% RSLogix 500 project Complex Boiler System.RSS, saved by version 8.30.00.16 %
PROJECT "UNTITLED"    % processor: Bul.1763 MicroLogix 1100 Series B %

PROGRAM FILES
  LAD 2 "MAIN"  10 rungs
  LAD 3 "DIGI IN"  11 rungs  % Digital Input Ladder Logic %
  LAD 4 "DIGI OUT"  4 rungs  % Digital Output Ladder Logic %
  LAD 5 "ANALOG IN"  5 rungs  % Analog Inout Ladder Logic %
  LAD 6 "ANALOG OUT"  2 rungs  % Analog Output Ladder Logic %
  LAD 7 "CONTROLS"  15 rungs
  LAD 8 "ALARMS"  28 rungs
  LAD 9 "DISPLAY"  2 rungs

DATA FILES
  O0 OUTPUT  9 elements
  I1 INPUT  16 elements
  S2 STATUS  66 elements
  B3 BINARY  5 elements
  T4 TIMER  13 elements
  C5 COUNTER  1 elements
  R6 CONTROL  1 elements
  N7 INTEGER  9 elements
  F8 FLOAT  1 elements
  PD9   1 elements

LADDER 2 "MAIN"
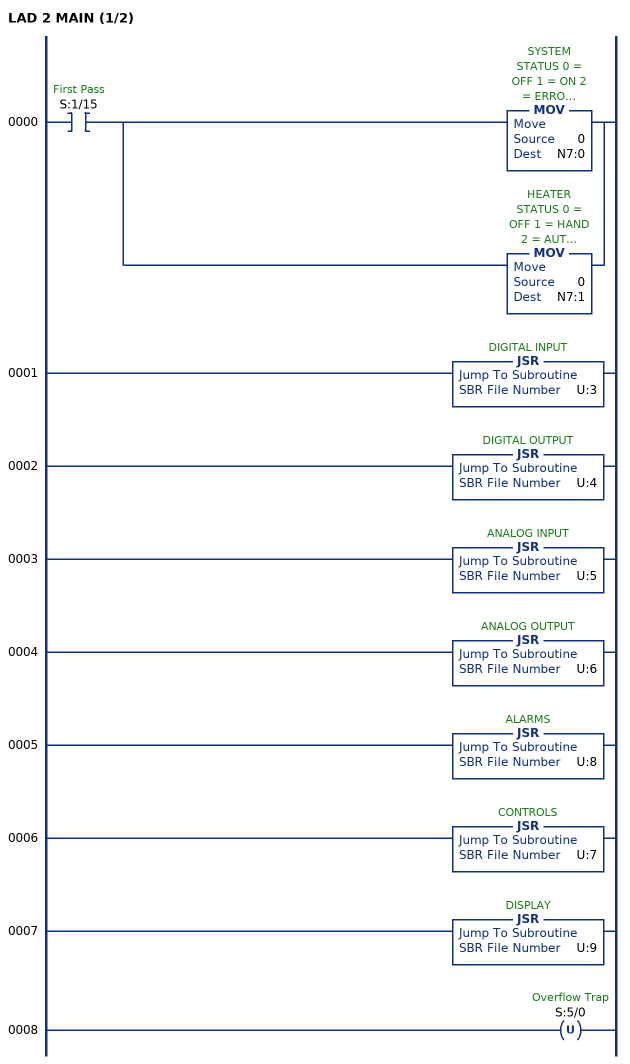
% Rung: 0 %
SOR XIC S:1/15 BST MOV 0 N7:0 NXB MOV 0 N7:1 BND EOR
%   S:1/15  "First Pass" %
%   N7:0  SYSTEM_STATUS  "SYSTEM STATUS 0 = OFF 1 = ON 2 = ERROR" %
%   N7:1  HEATER_STATUS  "HEATER STATUS 0 = OFF 1 = HAND 2 = AUTO" %
% Rung: 1 %
SOR JSR U:3 EOR
%   U:3  "DIGITAL INPUT" %
% Rung: 2 %
SOR JSR U:4 EOR
%   U:4  "DIGITAL OUTPUT" %
% Rung: 3 %
SOR JSR U:5 EOR
%   U:5  "ANALOG INPUT" %
% Rung: 4 %
SOR JSR U:6 EOR
%   U:6  "ANALOG OUTPUT" %
% Rung: 5 %
SOR JSR U:8 EOR
%   U:8  "ALARMS" %
% Rung: 6 %
SOR JSR U:7 EOR
%   U:7  "CONTROLS" %
% Rung: 7 %
SOR JSR U:9 EOR
%   U:9  "DISPLAY" %
% Rung: 8 %
SOR OTU S:5/0 EOR
%   S:5/0  "Overflow Trap" %

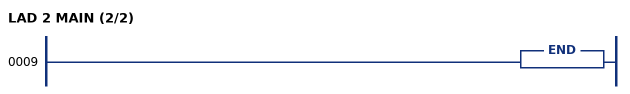
% Rung: 9 %
SOR END EOR

LADDER 3 "DIGI IN"    % Digital Input Ladder Logic %
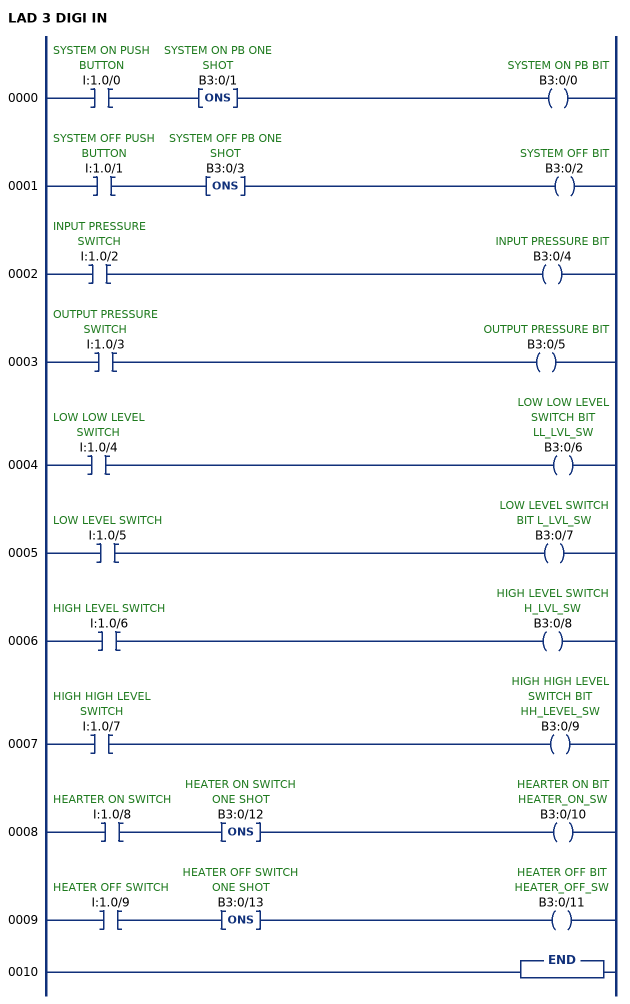
% Rung: 0 %
SOR XIC I:1.0/0 ONS B3:0/1 OTE B3:0/0 EOR
%   I:1.0/0  "SYSTEM ON PUSH BUTTON" %
%   B3:0/1  "SYSTEM ON PB ONE SHOT" %
%   B3:0/0  "SYSTEM ON PB BIT" %
% Rung: 1 %
SOR XIC I:1.0/1 ONS B3:0/3 OTE B3:0/2 EOR
%   I:1.0/1  "SYSTEM OFF PUSH BUTTON" %
%   B3:0/3  "SYSTEM OFF PB ONE SHOT" %
%   B3:0/2  "SYSTEM OFF BIT" %
% Rung: 2 %
SOR XIC I:1.0/2 OTE B3:0/4 EOR
%   I:1.0/2  "INPUT PRESSURE SWITCH" %
%   B3:0/4  "INPUT PRESSURE BIT" %
% Rung: 3 %
SOR XIC I:1.0/3 OTE B3:0/5 EOR
%   I:1.0/3  "OUTPUT PRESSURE SWITCH" %
%   B3:0/5  "OUTPUT PRESSURE BIT" %
% Rung: 4 %
SOR XIC I:1.0/4 OTE B3:0/6 EOR
%   I:1.0/4  "LOW LOW LEVEL SWITCH" %
%   B3:0/6  LL_LVL_SW  "LOW LOW LEVEL SWITCH BIT" %
% Rung: 5 %
SOR XIC I:1.0/5 OTE B3:0/7 EOR
%   I:1.0/5  "LOW LEVEL SWITCH" %
%   B3:0/7  L_LVL_SW  "LOW LEVEL SWITCH BIT" %
% Rung: 6 %
SOR XIC I:1.0/6 OTE B3:0/8 EOR
%   I:1.0/6  "HIGH LEVEL SWITCH" %
%   B3:0/8  H_LVL_SW  "HIGH LEVEL SWITCH" %
% Rung: 7 %
SOR XIC I:1.0/7 OTE B3:0/9 EOR
%   I:1.0/7  "HIGH HIGH LEVEL SWITCH" %
%   B3:0/9  HH_LEVEL_SW  "HIGH HIGH LEVEL SWITCH BIT" %
% Rung: 8 %
SOR XIC I:1.0/8 ONS B3:0/12 OTE B3:0/10 EOR
%   I:1.0/8  "HEARTER ON SWITCH" %
%   B3:0/12  "HEATER ON SWITCH ONE SHOT" %
%   B3:0/10  HEATER_ON_SW  "HEARTER ON BIT" %
% Rung: 9 %
SOR XIC I:1.0/9 ONS B3:0/13 OTE B3:0/11 EOR
%   I:1.0/9  "HEATER OFF SWITCH" %
%   B3:0/13  "HEATER OFF SWITCH ONE SHOT" %
%   B3:0/11  HEATER_OFF_SW  "HEATER OFF BIT" %
% Rung: 10 %
SOR END EOR

LADDER 4 "DIGI OUT"    % Digital Output Ladder Logic %
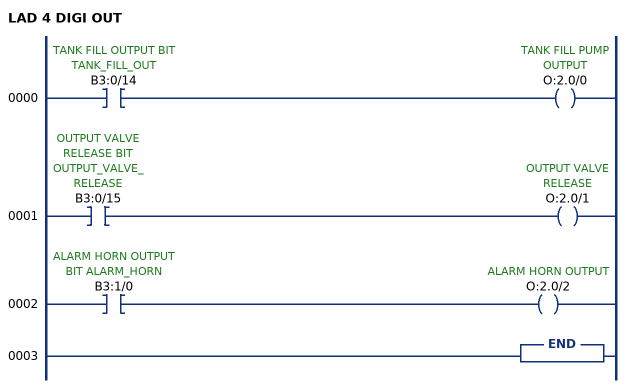
% Rung: 0 %
SOR XIC B3:0/14 OTE O:2.0/0 EOR
%   B3:0/14  TANK_FILL_OUT  "TANK FILL OUTPUT BIT" %
%   O:2.0/0  "TANK FILL PUMP OUTPUT" %
% Rung: 1 %
SOR XIC B3:0/15 OTE O:2.0/1 EOR
%   B3:0/15  OUTPUT_VALVE_RELEASE  "OUTPUT VALVE RELEASE BIT" %
%   O:2.0/1  "OUTPUT VALVE RELEASE" %
% Rung: 2 %
SOR XIC B3:1/0 OTE O:2.0/2 EOR
%   B3:1/0  ALARM_HORN  "ALARM HORN OUTPUT BIT" %
%   O:2.0/2  "ALARM HORN OUTPUT" %
% Rung: 3 %
SOR END EOR

LADDER 5 "ANALOG IN"    % Analog Inout Ladder Logic %
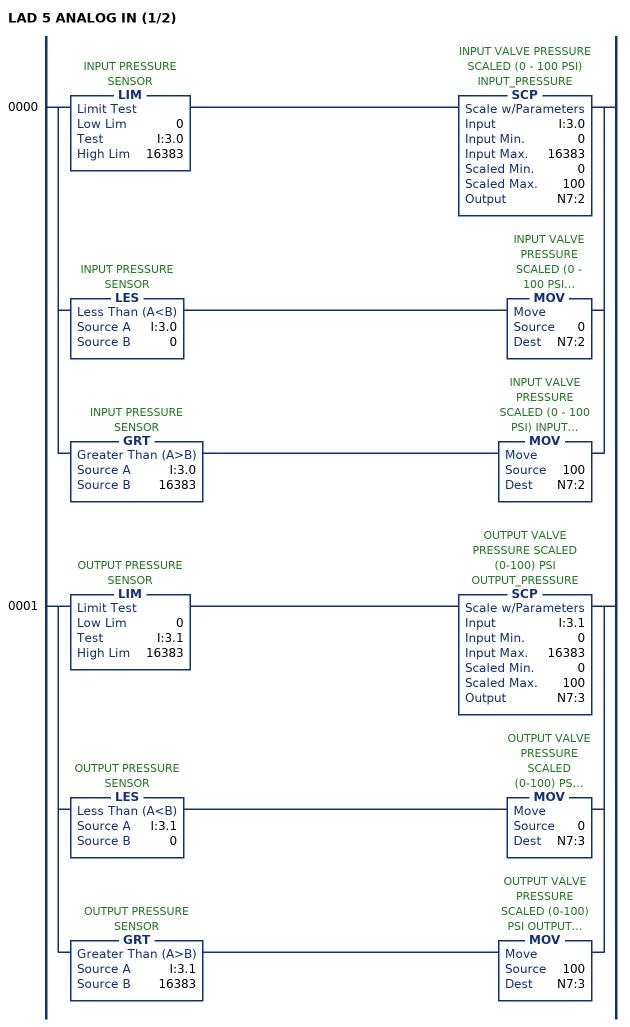
% Rung: 0 %
SOR BST LIM 0 I:3.0 16383 SCP I:3.0 0 16383 0 100 N7:2 NXB LES I:3.0 0 MOV 0 N7:2 NXB GRT I:3.0 16383 MOV 100 N7:2 BND EOR
%   I:3.0  "INPUT PRESSURE SENSOR" %
%   N7:2  INPUT_PRESSURE  "INPUT VALVE PRESSURE SCALED (0 - 100 PSI)" %
% Rung: 1 %
SOR BST LIM 0 I:3.1 16383 SCP I:3.1 0 16383 0 100 N7:3 NXB LES I:3.1 0 MOV 0 N7:3 NXB GRT I:3.1 16383 MOV 100 N7:3 BND EOR
%   I:3.1  "OUTPUT PRESSURE SENSOR" %
%   N7:3  OUTPUT_PRESSURE  "OUTPUT VALVE PRESSURE SCALED (0-100) PSI" %

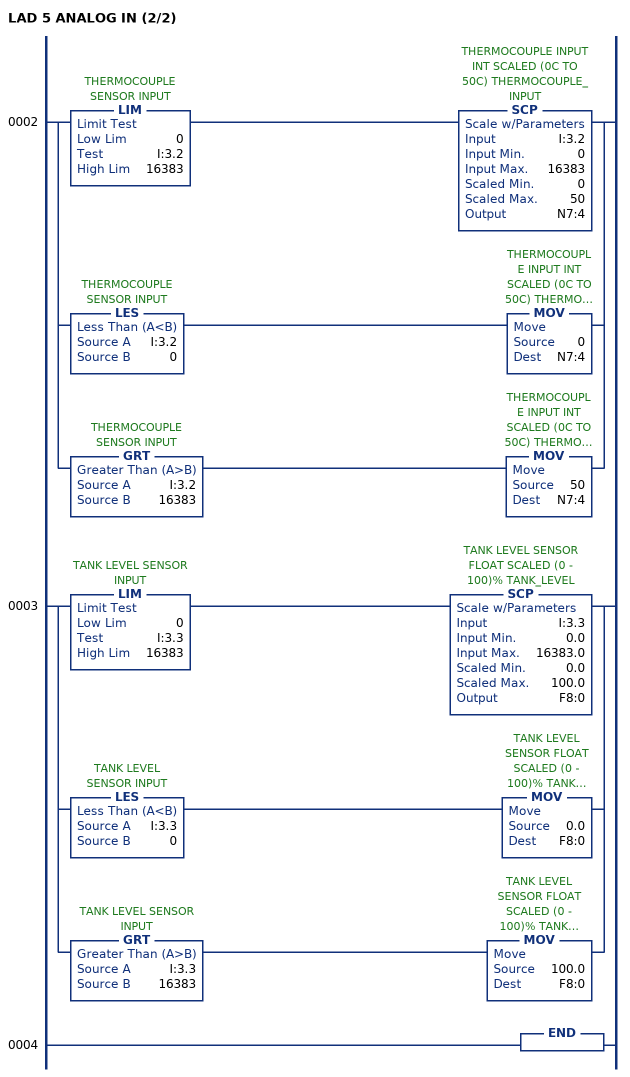
% Rung: 2 %
SOR BST LIM 0 I:3.2 16383 SCP I:3.2 0 16383 0 50 N7:4 NXB LES I:3.2 0 MOV 0 N7:4 NXB GRT I:3.2 16383 MOV 50 N7:4 BND EOR
%   I:3.2  "THERMOCOUPLE SENSOR INPUT" %
%   N7:4  THERMOCOUPLE_INPUT  "THERMOCOUPLE INPUT INT SCALED (0C TO 50C)" %
% Rung: 3 %
SOR BST LIM 0 I:3.3 16383 SCP I:3.3 0.0 16383.0 0.0 100.0 F8:0 NXB LES I:3.3 0 MOV 0.0 F8:0 NXB GRT I:3.3 16383 MOV 100.0 F8:0 BND EOR
%   I:3.3  "TANK LEVEL SENSOR INPUT" %
%   F8:0  TANK_LEVEL  "TANK LEVEL SENSOR FLOAT SCALED (0 - 100)%" %
% Rung: 4 %
SOR END EOR

LADDER 6 "ANALOG OUT"    % Analog Output Ladder Logic %
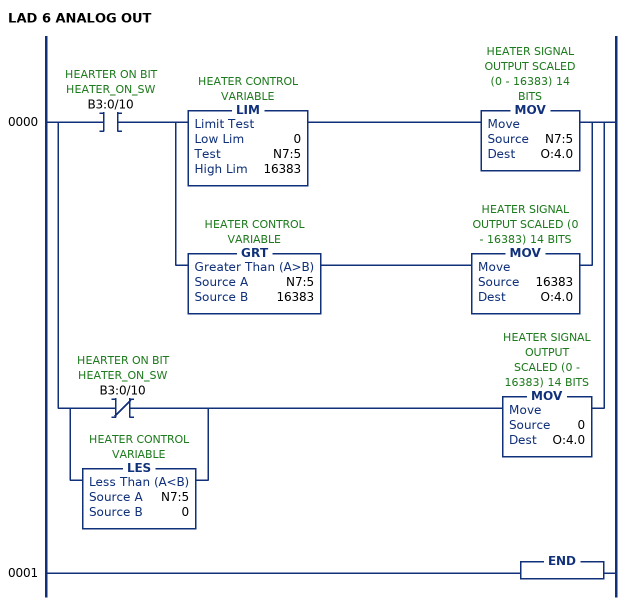
% Rung: 0 %
SOR BST XIC B3:0/10 BST LIM 0 N7:5 16383 MOV N7:5 O:4.0 NXB GRT N7:5 16383 MOV 16383 O:4.0 BND NXB BST XIO B3:0/10 NXB LES N7:5 0 BND MOV 0 O:4.0 BND EOR
%   B3:0/10  HEATER_ON_SW  "HEARTER ON BIT" %
%   N7:5  "HEATER CONTROL VARIABLE" %
%   O:4.0  "HEATER SIGNAL OUTPUT SCALED (0 - 16383) 14 BITS" %
% Rung: 1 %
SOR END EOR

LADDER 7 "CONTROLS"
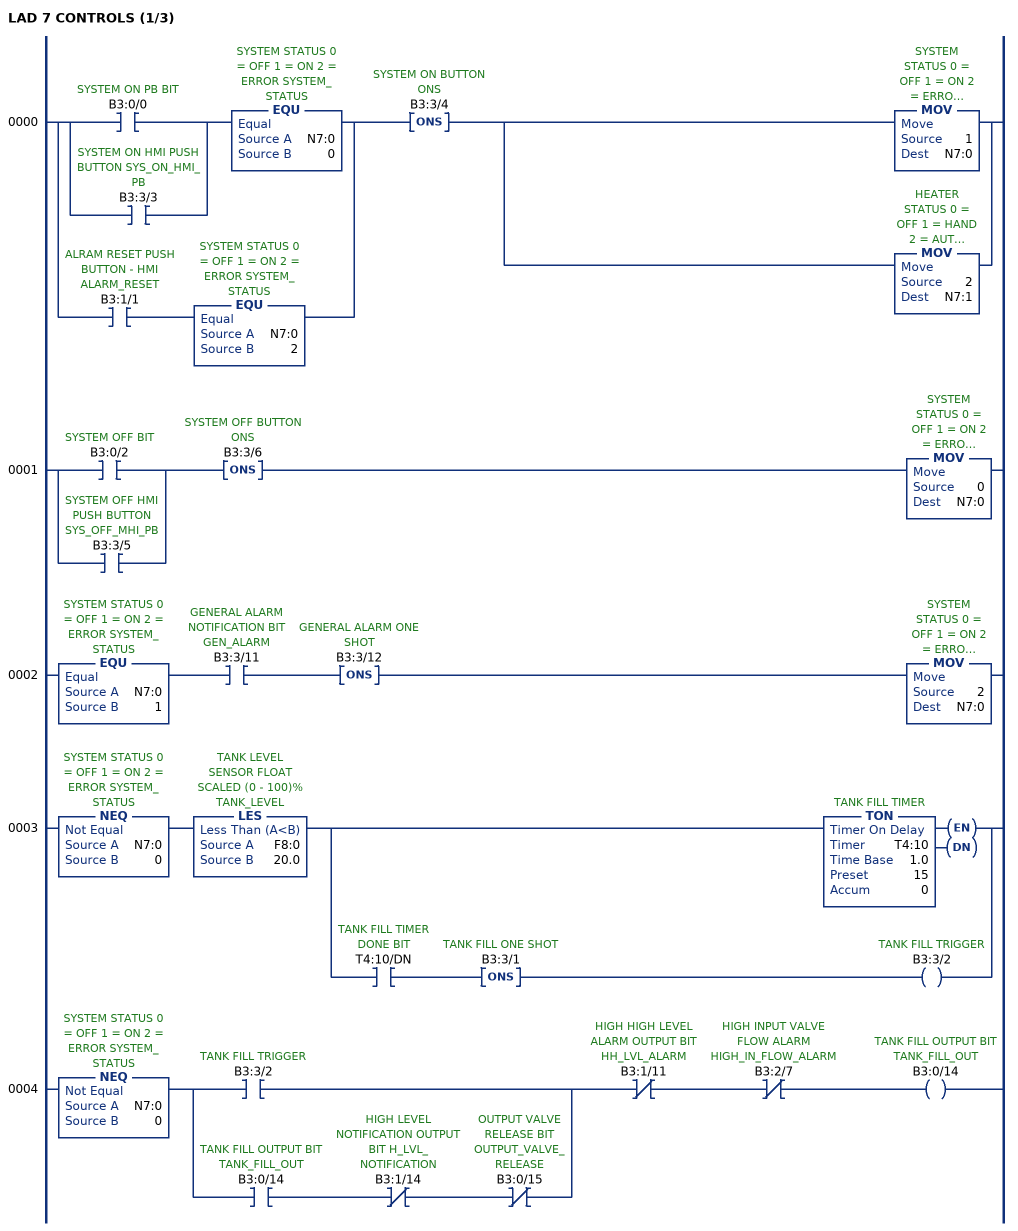
% Rung: 0 %
SOR BST BST XIC B3:0/0 NXB XIC B3:3/3 BND EQU N7:0 0 NXB XIC B3:1/1 EQU N7:0 2 BND ONS B3:3/4 BST MOV 1 N7:0 NXB MOV 2 N7:1 BND EOR
%   B3:0/0  "SYSTEM ON PB BIT" %
%   B3:3/3  SYS_ON_HMI_PB  "SYSTEM ON HMI PUSH BUTTON" %
%   N7:0  SYSTEM_STATUS  "SYSTEM STATUS 0 = OFF 1 = ON 2 = ERROR" %
%   B3:1/1  ALARM_RESET  "ALRAM RESET PUSH BUTTON - HMI" %
%   B3:3/4  "SYSTEM ON BUTTON ONS" %
%   N7:1  HEATER_STATUS  "HEATER STATUS 0 = OFF 1 = HAND 2 = AUTO" %
% Rung: 1 %
SOR BST XIC B3:0/2 NXB XIC B3:3/5 BND ONS B3:3/6 MOV 0 N7:0 EOR
%   B3:0/2  "SYSTEM OFF BIT" %
%   B3:3/5  SYS_OFF_MHI_PB  "SYSTEM OFF HMI PUSH BUTTON" %
%   B3:3/6  "SYSTEM OFF BUTTON ONS" %
%   N7:0  SYSTEM_STATUS  "SYSTEM STATUS 0 = OFF 1 = ON 2 = ERROR" %
% Rung: 2 %
SOR EQU N7:0 1 XIC B3:3/11 ONS B3:3/12 MOV 2 N7:0 EOR
%   N7:0  SYSTEM_STATUS  "SYSTEM STATUS 0 = OFF 1 = ON 2 = ERROR" %
%   B3:3/11  GEN_ALARM  "GENERAL ALARM NOTIFICATION BIT" %
%   B3:3/12  "GENERAL ALARM ONE SHOT" %
% Rung: 3 %
SOR NEQ N7:0 0 LES F8:0 20.0 BST TON T4:10 1.0 15 0 NXB XIC T4:10/DN ONS B3:3/1 OTE B3:3/2 BND EOR
%   N7:0  SYSTEM_STATUS  "SYSTEM STATUS 0 = OFF 1 = ON 2 = ERROR" %
%   F8:0  TANK_LEVEL  "TANK LEVEL SENSOR FLOAT SCALED (0 - 100)%" %
%   T4:10  "TANK FILL TIMER" %
%   T4:10/DN  "TANK FILL TIMER DONE BIT" %
%   B3:3/1  "TANK FILL ONE SHOT" %
%   B3:3/2  "TANK FILL TRIGGER" %
% Rung: 4 %
SOR NEQ N7:0 0 BST XIC B3:3/2 NXB XIC B3:0/14 XIO B3:1/14 XIO B3:0/15 BND XIO B3:1/11 XIO B3:2/7 OTE B3:0/14 EOR
%   N7:0  SYSTEM_STATUS  "SYSTEM STATUS 0 = OFF 1 = ON 2 = ERROR" %
%   B3:3/2  "TANK FILL TRIGGER" %
%   B3:0/14  TANK_FILL_OUT  "TANK FILL OUTPUT BIT" %
%   B3:1/14  H_LVL_NOTIFICATION  "HIGH LEVEL NOTIFICATION OUTPUT BIT" %
%   B3:0/15  OUTPUT_VALVE_RELEASE  "OUTPUT VALVE RELEASE BIT" %
%   B3:1/11  HH_LVL_ALARM  "HIGH HIGH LEVEL ALARM OUTPUT BIT" %
%   B3:2/7  HIGH_IN_FLOW_ALARM  "HIGH INPUT VALVE FLOW ALARM" %

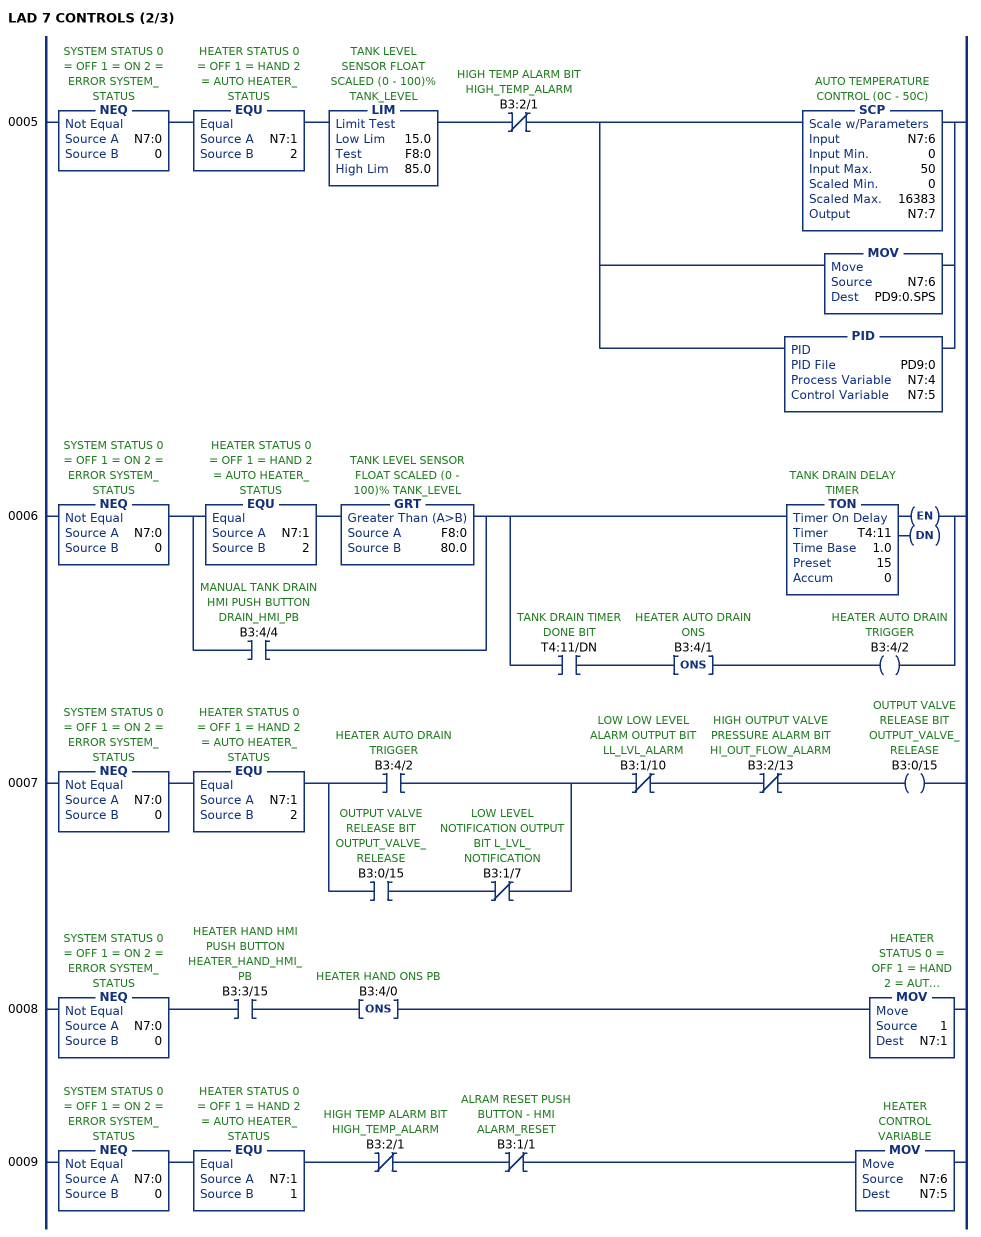
% Rung: 5 %
SOR NEQ N7:0 0 EQU N7:1 2 LIM 15.0 F8:0 85.0 XIO B3:2/1 BST SCP N7:6 0 50 0 16383 N7:7 NXB MOV N7:6 PD9:0.SPS NXB PID PD9:0 N7:4 N7:5 BND EOR
%   N7:0  SYSTEM_STATUS  "SYSTEM STATUS 0 = OFF 1 = ON 2 = ERROR" %
%   N7:1  HEATER_STATUS  "HEATER STATUS 0 = OFF 1 = HAND 2 = AUTO" %
%   F8:0  TANK_LEVEL  "TANK LEVEL SENSOR FLOAT SCALED (0 - 100)%" %
%   B3:2/1  HIGH_TEMP_ALARM  "HIGH TEMP ALARM BIT" %
%   N7:6  "AUTO TEMPERATURE CONTROL SCALED(0 - 16383)" %
%   N7:7  "AUTO TEMPERATURE CONTROL (0C - 50C)" %
%   N7:4  THERMOCOUPLE_INPUT  "THERMOCOUPLE INPUT INT SCALED (0C TO 50C)" %
%   N7:5  "HEATER CONTROL VARIABLE" %
% Rung: 6 %
SOR NEQ N7:0 0 BST EQU N7:1 2 GRT F8:0 80.0 NXB XIC B3:4/4 BND BST TON T4:11 1.0 15 0 NXB XIC T4:11/DN ONS B3:4/1 OTE B3:4/2 BND EOR
%   N7:0  SYSTEM_STATUS  "SYSTEM STATUS 0 = OFF 1 = ON 2 = ERROR" %
%   N7:1  HEATER_STATUS  "HEATER STATUS 0 = OFF 1 = HAND 2 = AUTO" %
%   F8:0  TANK_LEVEL  "TANK LEVEL SENSOR FLOAT SCALED (0 - 100)%" %
%   B3:4/4  DRAIN_HMI_PB  "MANUAL TANK DRAIN HMI PUSH BUTTON" %
%   T4:11  "TANK DRAIN DELAY TIMER" %
%   T4:11/DN  "TANK DRAIN TIMER DONE BIT" %
%   B3:4/1  "HEATER AUTO DRAIN ONS" %
%   B3:4/2  "HEATER AUTO DRAIN TRIGGER" %
% Rung: 7 %
SOR NEQ N7:0 0 EQU N7:1 2 BST XIC B3:4/2 NXB XIC B3:0/15 XIO B3:1/7 BND XIO B3:1/10 XIO B3:2/13 OTE B3:0/15 EOR
%   N7:0  SYSTEM_STATUS  "SYSTEM STATUS 0 = OFF 1 = ON 2 = ERROR" %
%   N7:1  HEATER_STATUS  "HEATER STATUS 0 = OFF 1 = HAND 2 = AUTO" %
%   B3:4/2  "HEATER AUTO DRAIN TRIGGER" %
%   B3:0/15  OUTPUT_VALVE_RELEASE  "OUTPUT VALVE RELEASE BIT" %
%   B3:1/7  L_LVL_NOTIFICATION  "LOW LEVEL NOTIFICATION OUTPUT BIT" %
%   B3:1/10  LL_LVL_ALARM  "LOW LOW LEVEL ALARM OUTPUT BIT" %
%   B3:2/13  HI_OUT_FLOW_ALARM  "HIGH OUTPUT VALVE PRESSURE ALARM BIT" %
% Rung: 8 %
SOR NEQ N7:0 0 XIC B3:3/15 ONS B3:4/0 MOV 1 N7:1 EOR
%   N7:0  SYSTEM_STATUS  "SYSTEM STATUS 0 = OFF 1 = ON 2 = ERROR" %
%   B3:3/15  HEATER_HAND_HMI_PB  "HEATER HAND HMI PUSH BUTTON" %
%   B3:4/0  "HEATER HAND ONS PB" %
%   N7:1  HEATER_STATUS  "HEATER STATUS 0 = OFF 1 = HAND 2 = AUTO" %
% Rung: 9 %
SOR NEQ N7:0 0 EQU N7:1 1 XIO B3:2/1 XIO B3:1/1 MOV N7:6 N7:5 EOR
%   N7:0  SYSTEM_STATUS  "SYSTEM STATUS 0 = OFF 1 = ON 2 = ERROR" %
%   N7:1  HEATER_STATUS  "HEATER STATUS 0 = OFF 1 = HAND 2 = AUTO" %
%   B3:2/1  HIGH_TEMP_ALARM  "HIGH TEMP ALARM BIT" %
%   B3:1/1  ALARM_RESET  "ALRAM RESET PUSH BUTTON - HMI" %
%   N7:6  "AUTO TEMPERATURE CONTROL SCALED(0 - 16383)" %
%   N7:5  "HEATER CONTROL VARIABLE" %

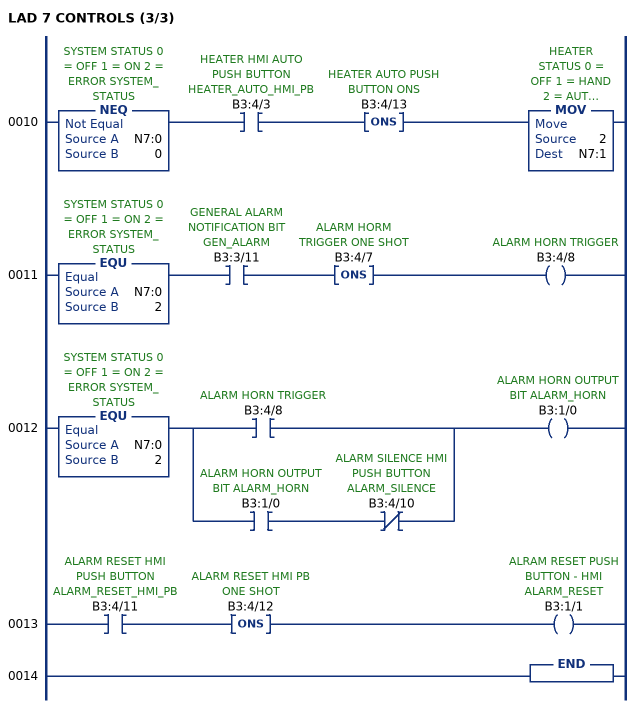
% Rung: 10 %
SOR NEQ N7:0 0 XIC B3:4/3 ONS B3:4/13 MOV 2 N7:1 EOR
%   N7:0  SYSTEM_STATUS  "SYSTEM STATUS 0 = OFF 1 = ON 2 = ERROR" %
%   B3:4/3  HEATER_AUTO_HMI_PB  "HEATER HMI AUTO PUSH BUTTON" %
%   B3:4/13  "HEATER AUTO PUSH BUTTON ONS" %
%   N7:1  HEATER_STATUS  "HEATER STATUS 0 = OFF 1 = HAND 2 = AUTO" %
% Rung: 11 %
SOR EQU N7:0 2 XIC B3:3/11 ONS B3:4/7 OTE B3:4/8 EOR
%   N7:0  SYSTEM_STATUS  "SYSTEM STATUS 0 = OFF 1 = ON 2 = ERROR" %
%   B3:3/11  GEN_ALARM  "GENERAL ALARM NOTIFICATION BIT" %
%   B3:4/7  "ALARM HORM TRIGGER ONE SHOT" %
%   B3:4/8  "ALARM HORN TRIGGER" %
% Rung: 12 %
SOR EQU N7:0 2 BST XIC B3:4/8 NXB XIC B3:1/0 XIO B3:4/10 BND OTE B3:1/0 EOR
%   N7:0  SYSTEM_STATUS  "SYSTEM STATUS 0 = OFF 1 = ON 2 = ERROR" %
%   B3:4/8  "ALARM HORN TRIGGER" %
%   B3:1/0  ALARM_HORN  "ALARM HORN OUTPUT BIT" %
%   B3:4/10  ALARM_SILENCE  "ALARM SILENCE HMI PUSH BUTTON" %
% Rung: 13 %
SOR XIC B3:4/11 ONS B3:4/12 OTE B3:1/1 EOR
%   B3:4/11  ALARM_RESET_HMI_PB  "ALARM RESET HMI PUSH BUTTON" %
%   B3:4/12  "ALARM RESET HMI PB ONE SHOT" %
%   B3:1/1  ALARM_RESET  "ALRAM RESET PUSH BUTTON - HMI" %
% Rung: 14 %
SOR END EOR

LADDER 8 "ALARMS"
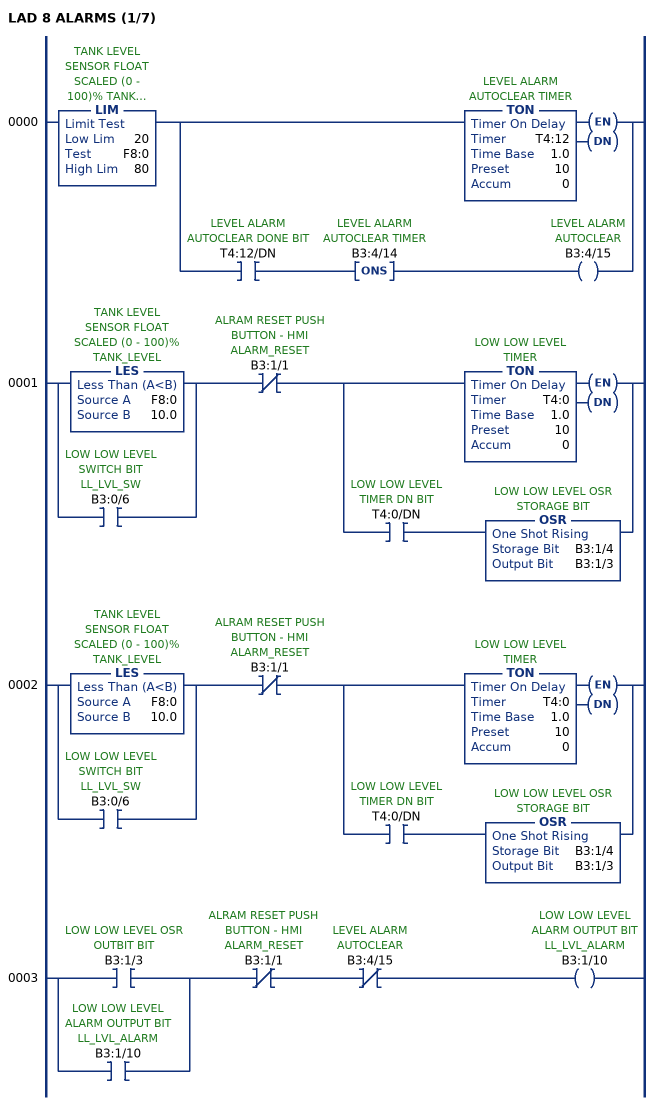
% Rung: 0 %
SOR LIM 20 F8:0 80 BST TON T4:12 1.0 10 0 NXB XIC T4:12/DN ONS B3:4/14 OTE B3:4/15 BND EOR
%   F8:0  TANK_LEVEL  "TANK LEVEL SENSOR FLOAT SCALED (0 - 100)%" %
%   T4:12  "LEVEL ALARM AUTOCLEAR TIMER" %
%   T4:12/DN  "LEVEL ALARM AUTOCLEAR DONE BIT" %
%   B3:4/14  "LEVEL ALARM AUTOCLEAR TIMER" %
%   B3:4/15  "LEVEL ALARM AUTOCLEAR" %
% Rung: 1 %
SOR BST LES F8:0 10.0 NXB XIC B3:0/6 BND XIO B3:1/1 BST TON T4:0 1.0 10 0 NXB XIC T4:0/DN OSR B3:1/4 B3:1/3 BND EOR
%   F8:0  TANK_LEVEL  "TANK LEVEL SENSOR FLOAT SCALED (0 - 100)%" %
%   B3:0/6  LL_LVL_SW  "LOW LOW LEVEL SWITCH BIT" %
%   B3:1/1  ALARM_RESET  "ALRAM RESET PUSH BUTTON - HMI" %
%   T4:0  "LOW LOW LEVEL TIMER" %
%   T4:0/DN  "LOW LOW LEVEL TIMER DN BIT" %
%   B3:1/4  "LOW LOW LEVEL OSR STORAGE BIT" %
%   B3:1/3  "LOW LOW LEVEL OSR OUTBIT BIT" %
% Rung: 2 %
SOR BST LES F8:0 10.0 NXB XIC B3:0/6 BND XIO B3:1/1 BST TON T4:0 1.0 10 0 NXB XIC T4:0/DN OSR B3:1/4 B3:1/3 BND EOR
%   F8:0  TANK_LEVEL  "TANK LEVEL SENSOR FLOAT SCALED (0 - 100)%" %
%   B3:0/6  LL_LVL_SW  "LOW LOW LEVEL SWITCH BIT" %
%   B3:1/1  ALARM_RESET  "ALRAM RESET PUSH BUTTON - HMI" %
%   T4:0  "LOW LOW LEVEL TIMER" %
%   T4:0/DN  "LOW LOW LEVEL TIMER DN BIT" %
%   B3:1/4  "LOW LOW LEVEL OSR STORAGE BIT" %
%   B3:1/3  "LOW LOW LEVEL OSR OUTBIT BIT" %
% Rung: 3 %
SOR BST XIC B3:1/3 NXB XIC B3:1/10 BND XIO B3:1/1 XIO B3:4/15 OTE B3:1/10 EOR
%   B3:1/3  "LOW LOW LEVEL OSR OUTBIT BIT" %
%   B3:1/10  LL_LVL_ALARM  "LOW LOW LEVEL ALARM OUTPUT BIT" %
%   B3:1/1  ALARM_RESET  "ALRAM RESET PUSH BUTTON - HMI" %
%   B3:4/15  "LEVEL ALARM AUTOCLEAR" %

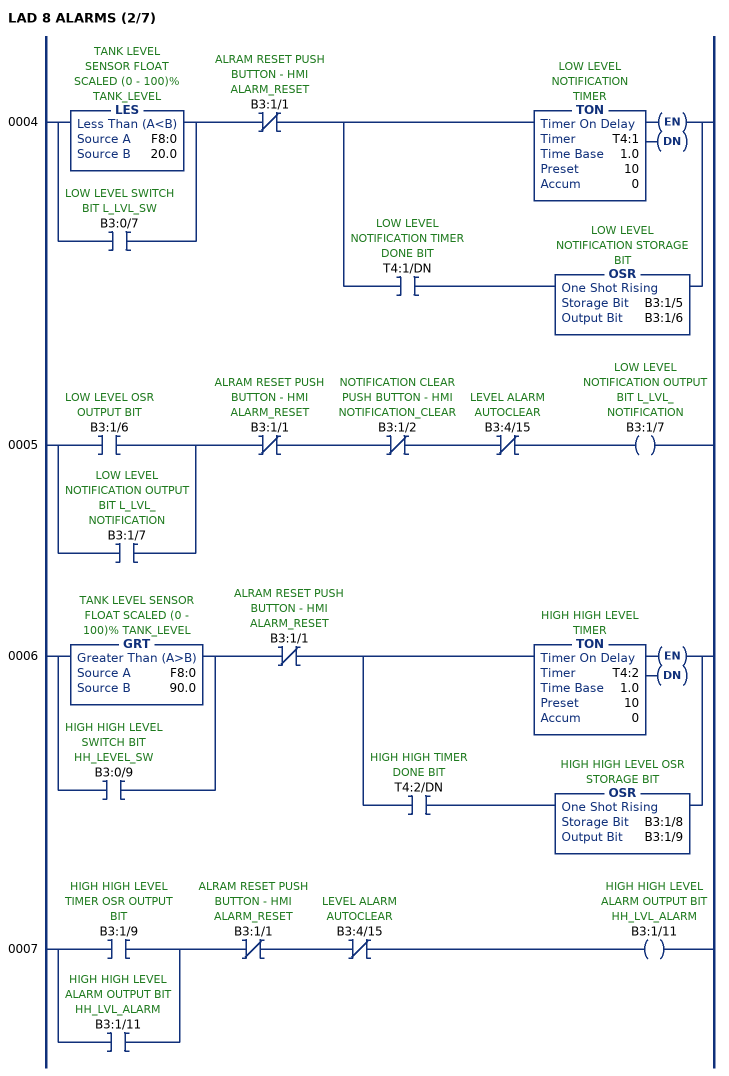
% Rung: 4 %
SOR BST LES F8:0 20.0 NXB XIC B3:0/7 BND XIO B3:1/1 BST TON T4:1 1.0 10 0 NXB XIC T4:1/DN OSR B3:1/5 B3:1/6 BND EOR
%   F8:0  TANK_LEVEL  "TANK LEVEL SENSOR FLOAT SCALED (0 - 100)%" %
%   B3:0/7  L_LVL_SW  "LOW LEVEL SWITCH BIT" %
%   B3:1/1  ALARM_RESET  "ALRAM RESET PUSH BUTTON - HMI" %
%   T4:1  "LOW LEVEL NOTIFICATION TIMER" %
%   T4:1/DN  "LOW LEVEL NOTIFICATION TIMER DONE BIT" %
%   B3:1/5  "LOW LEVEL NOTIFICATION STORAGE BIT" %
%   B3:1/6  "LOW LEVEL OSR OUTPUT BIT" %
% Rung: 5 %
SOR BST XIC B3:1/6 NXB XIC B3:1/7 BND XIO B3:1/1 XIO B3:1/2 XIO B3:4/15 OTE B3:1/7 EOR
%   B3:1/6  "LOW LEVEL OSR OUTPUT BIT" %
%   B3:1/7  L_LVL_NOTIFICATION  "LOW LEVEL NOTIFICATION OUTPUT BIT" %
%   B3:1/1  ALARM_RESET  "ALRAM RESET PUSH BUTTON - HMI" %
%   B3:1/2  NOTIFICATION_CLEAR  "NOTIFICATION CLEAR PUSH BUTTON - HMI" %
%   B3:4/15  "LEVEL ALARM AUTOCLEAR" %
% Rung: 6 %
SOR BST GRT F8:0 90.0 NXB XIC B3:0/9 BND XIO B3:1/1 BST TON T4:2 1.0 10 0 NXB XIC T4:2/DN OSR B3:1/8 B3:1/9 BND EOR
%   F8:0  TANK_LEVEL  "TANK LEVEL SENSOR FLOAT SCALED (0 - 100)%" %
%   B3:0/9  HH_LEVEL_SW  "HIGH HIGH LEVEL SWITCH BIT" %
%   B3:1/1  ALARM_RESET  "ALRAM RESET PUSH BUTTON - HMI" %
%   T4:2  "HIGH HIGH LEVEL TIMER" %
%   T4:2/DN  "HIGH HIGH TIMER DONE BIT" %
%   B3:1/8  "HIGH HIGH LEVEL OSR STORAGE BIT" %
%   B3:1/9  "HIGH HIGH LEVEL TIMER OSR OUTPUT BIT" %
% Rung: 7 %
SOR BST XIC B3:1/9 NXB XIC B3:1/11 BND XIO B3:1/1 XIO B3:4/15 OTE B3:1/11 EOR
%   B3:1/9  "HIGH HIGH LEVEL TIMER OSR OUTPUT BIT" %
%   B3:1/11  HH_LVL_ALARM  "HIGH HIGH LEVEL ALARM OUTPUT BIT" %
%   B3:1/1  ALARM_RESET  "ALRAM RESET PUSH BUTTON - HMI" %
%   B3:4/15  "LEVEL ALARM AUTOCLEAR" %

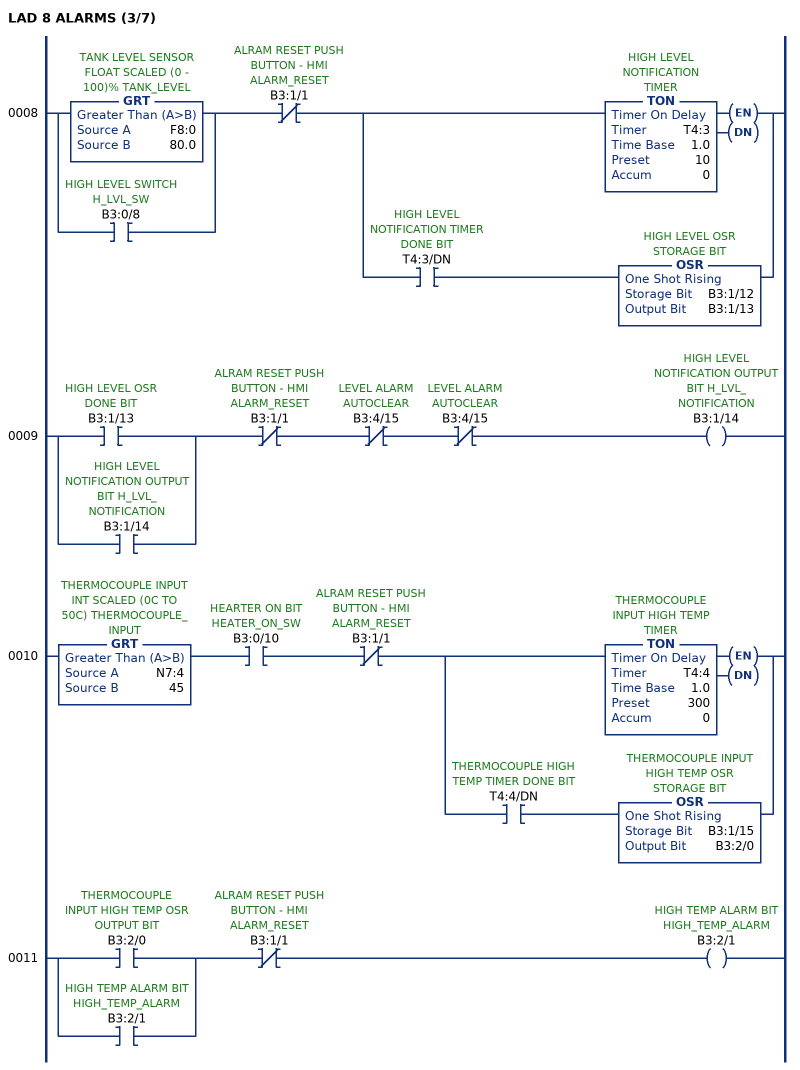
% Rung: 8 %
SOR BST GRT F8:0 80.0 NXB XIC B3:0/8 BND XIO B3:1/1 BST TON T4:3 1.0 10 0 NXB XIC T4:3/DN OSR B3:1/12 B3:1/13 BND EOR
%   F8:0  TANK_LEVEL  "TANK LEVEL SENSOR FLOAT SCALED (0 - 100)%" %
%   B3:0/8  H_LVL_SW  "HIGH LEVEL SWITCH" %
%   B3:1/1  ALARM_RESET  "ALRAM RESET PUSH BUTTON - HMI" %
%   T4:3  "HIGH LEVEL NOTIFICATION TIMER" %
%   T4:3/DN  "HIGH LEVEL NOTIFICATION TIMER DONE BIT" %
%   B3:1/12  "HIGH LEVEL OSR STORAGE BIT" %
%   B3:1/13  "HIGH LEVEL OSR DONE BIT" %
% Rung: 9 %
SOR BST XIC B3:1/13 NXB XIC B3:1/14 BND XIO B3:1/1 XIO B3:4/15 XIO B3:4/15 OTE B3:1/14 EOR
%   B3:1/13  "HIGH LEVEL OSR DONE BIT" %
%   B3:1/14  H_LVL_NOTIFICATION  "HIGH LEVEL NOTIFICATION OUTPUT BIT" %
%   B3:1/1  ALARM_RESET  "ALRAM RESET PUSH BUTTON - HMI" %
%   B3:4/15  "LEVEL ALARM AUTOCLEAR" %
% Rung: 10 %
SOR GRT N7:4 45 XIC B3:0/10 XIO B3:1/1 BST TON T4:4 1.0 300 0 NXB XIC T4:4/DN OSR B3:1/15 B3:2/0 BND EOR
%   N7:4  THERMOCOUPLE_INPUT  "THERMOCOUPLE INPUT INT SCALED (0C TO 50C)" %
%   B3:0/10  HEATER_ON_SW  "HEARTER ON BIT" %
%   B3:1/1  ALARM_RESET  "ALRAM RESET PUSH BUTTON - HMI" %
%   T4:4  "THERMOCOUPLE INPUT HIGH TEMP TIMER" %
%   T4:4/DN  "THERMOCOUPLE HIGH TEMP TIMER DONE BIT" %
%   B3:1/15  "THERMOCOUPLE INPUT HIGH TEMP OSR STORAGE BIT" %
%   B3:2/0  "THERMOCOUPLE INPUT HIGH TEMP OSR OUTPUT BIT" %
% Rung: 11 %
SOR BST XIC B3:2/0 NXB XIC B3:2/1 BND XIO B3:1/1 OTE B3:2/1 EOR
%   B3:2/0  "THERMOCOUPLE INPUT HIGH TEMP OSR OUTPUT BIT" %
%   B3:2/1  HIGH_TEMP_ALARM  "HIGH TEMP ALARM BIT" %
%   B3:1/1  ALARM_RESET  "ALRAM RESET PUSH BUTTON - HMI" %

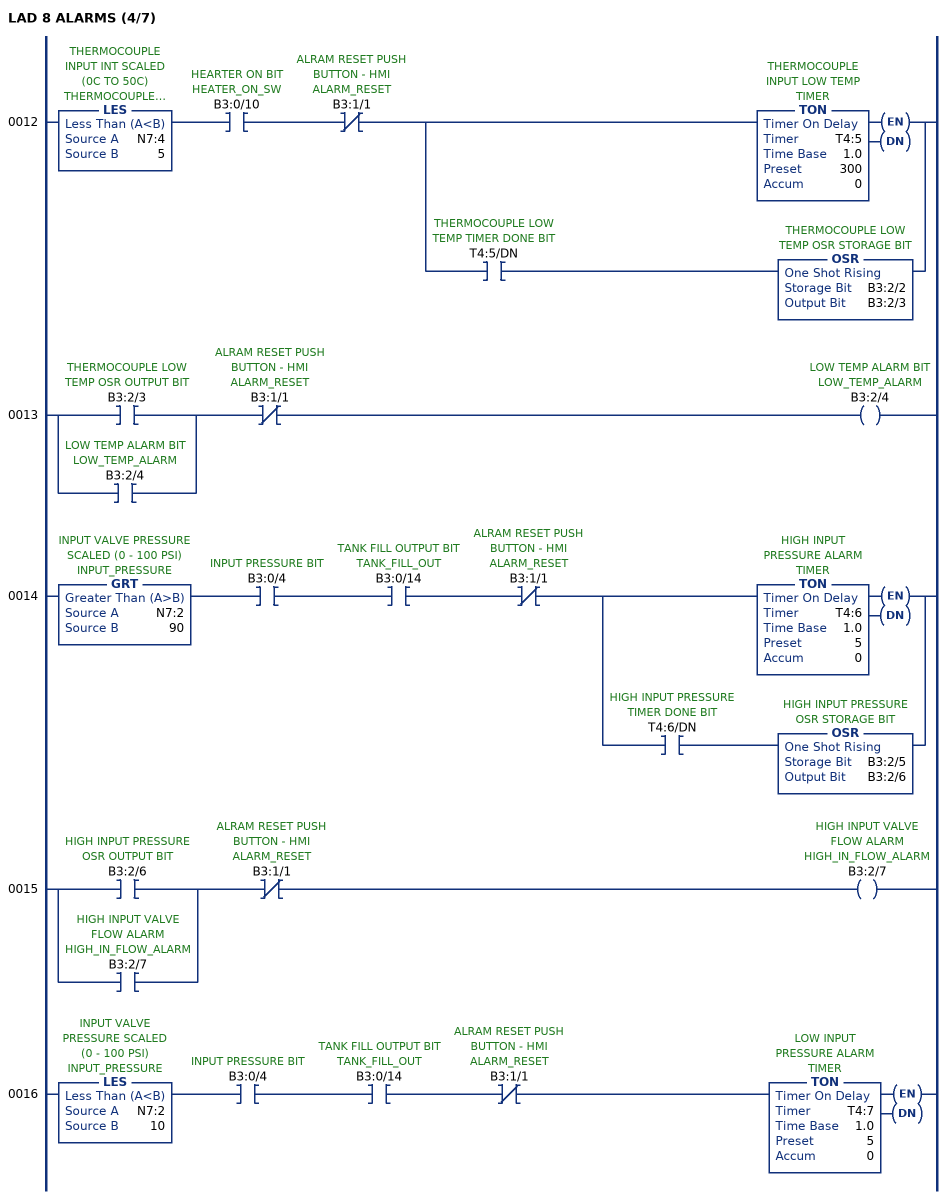
% Rung: 12 %
SOR LES N7:4 5 XIC B3:0/10 XIO B3:1/1 BST TON T4:5 1.0 300 0 NXB XIC T4:5/DN OSR B3:2/2 B3:2/3 BND EOR
%   N7:4  THERMOCOUPLE_INPUT  "THERMOCOUPLE INPUT INT SCALED (0C TO 50C)" %
%   B3:0/10  HEATER_ON_SW  "HEARTER ON BIT" %
%   B3:1/1  ALARM_RESET  "ALRAM RESET PUSH BUTTON - HMI" %
%   T4:5  "THERMOCOUPLE INPUT LOW TEMP TIMER" %
%   T4:5/DN  "THERMOCOUPLE LOW TEMP TIMER DONE BIT" %
%   B3:2/2  "THERMOCOUPLE LOW TEMP OSR STORAGE BIT" %
%   B3:2/3  "THERMOCOUPLE LOW TEMP OSR OUTPUT BIT" %
% Rung: 13 %
SOR BST XIC B3:2/3 NXB XIC B3:2/4 BND XIO B3:1/1 OTE B3:2/4 EOR
%   B3:2/3  "THERMOCOUPLE LOW TEMP OSR OUTPUT BIT" %
%   B3:2/4  LOW_TEMP_ALARM  "LOW TEMP ALARM BIT" %
%   B3:1/1  ALARM_RESET  "ALRAM RESET PUSH BUTTON - HMI" %
% Rung: 14 %
SOR GRT N7:2 90 XIC B3:0/4 XIC B3:0/14 XIO B3:1/1 BST TON T4:6 1.0 5 0 NXB XIC T4:6/DN OSR B3:2/5 B3:2/6 BND EOR
%   N7:2  INPUT_PRESSURE  "INPUT VALVE PRESSURE SCALED (0 - 100 PSI)" %
%   B3:0/4  "INPUT PRESSURE BIT" %
%   B3:0/14  TANK_FILL_OUT  "TANK FILL OUTPUT BIT" %
%   B3:1/1  ALARM_RESET  "ALRAM RESET PUSH BUTTON - HMI" %
%   T4:6  "HIGH INPUT PRESSURE ALARM TIMER" %
%   T4:6/DN  "HIGH INPUT PRESSURE TIMER DONE BIT" %
%   B3:2/5  "HIGH INPUT PRESSURE OSR STORAGE BIT" %
%   B3:2/6  "HIGH INPUT PRESSURE OSR OUTPUT BIT" %
% Rung: 15 %
SOR BST XIC B3:2/6 NXB XIC B3:2/7 BND XIO B3:1/1 OTE B3:2/7 EOR
%   B3:2/6  "HIGH INPUT PRESSURE OSR OUTPUT BIT" %
%   B3:2/7  HIGH_IN_FLOW_ALARM  "HIGH INPUT VALVE FLOW ALARM" %
%   B3:1/1  ALARM_RESET  "ALRAM RESET PUSH BUTTON - HMI" %
% Rung: 16 %
SOR LES N7:2 10 XIC B3:0/4 XIC B3:0/14 XIO B3:1/1 TON T4:7 1.0 5 0 EOR
%   N7:2  INPUT_PRESSURE  "INPUT VALVE PRESSURE SCALED (0 - 100 PSI)" %
%   B3:0/4  "INPUT PRESSURE BIT" %
%   B3:0/14  TANK_FILL_OUT  "TANK FILL OUTPUT BIT" %
%   B3:1/1  ALARM_RESET  "ALRAM RESET PUSH BUTTON - HMI" %
%   T4:7  "LOW INPUT PRESSURE ALARM TIMER" %

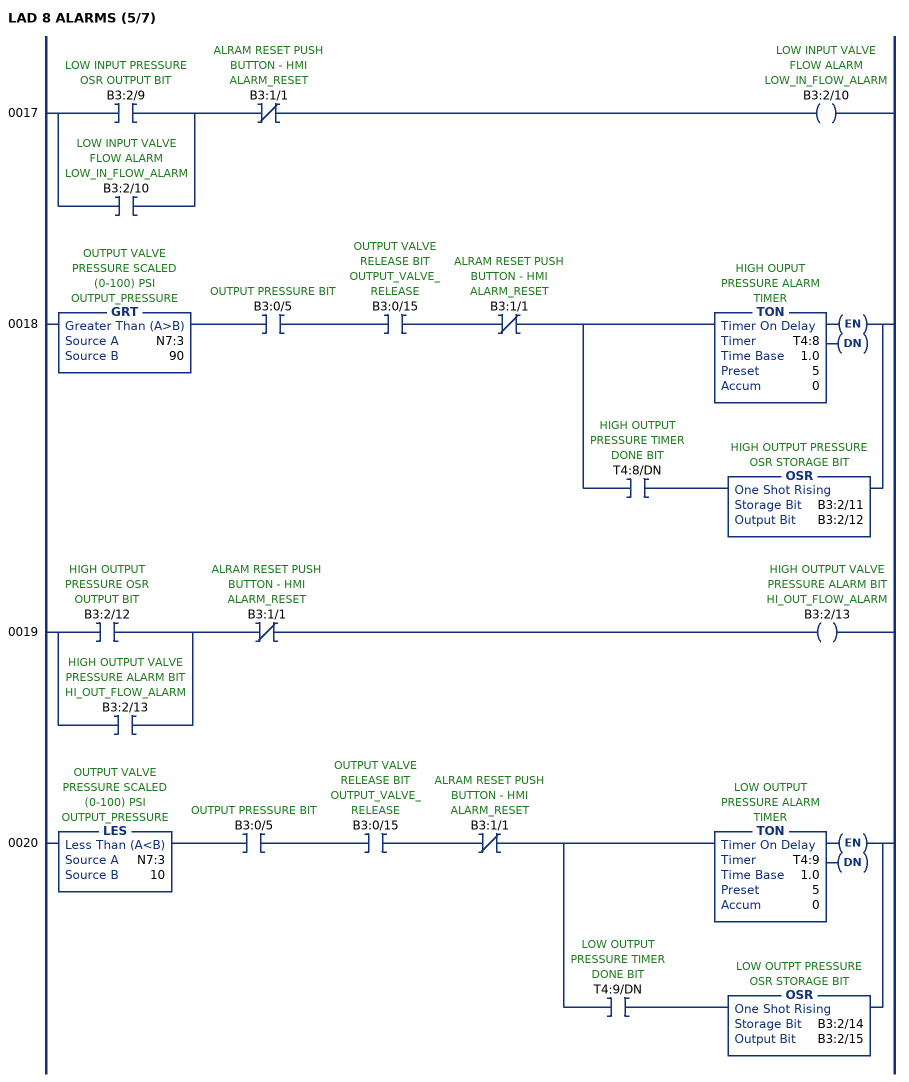
% Rung: 17 %
SOR BST XIC B3:2/9 NXB XIC B3:2/10 BND XIO B3:1/1 OTE B3:2/10 EOR
%   B3:2/9  "LOW INPUT PRESSURE OSR OUTPUT BIT" %
%   B3:2/10  LOW_IN_FLOW_ALARM  "LOW INPUT VALVE FLOW ALARM" %
%   B3:1/1  ALARM_RESET  "ALRAM RESET PUSH BUTTON - HMI" %
% Rung: 18 %
SOR GRT N7:3 90 XIC B3:0/5 XIC B3:0/15 XIO B3:1/1 BST TON T4:8 1.0 5 0 NXB XIC T4:8/DN OSR B3:2/11 B3:2/12 BND EOR
%   N7:3  OUTPUT_PRESSURE  "OUTPUT VALVE PRESSURE SCALED (0-100) PSI" %
%   B3:0/5  "OUTPUT PRESSURE BIT" %
%   B3:0/15  OUTPUT_VALVE_RELEASE  "OUTPUT VALVE RELEASE BIT" %
%   B3:1/1  ALARM_RESET  "ALRAM RESET PUSH BUTTON - HMI" %
%   T4:8  "HIGH OUPUT PRESSURE ALARM TIMER" %
%   T4:8/DN  "HIGH OUTPUT PRESSURE TIMER DONE BIT" %
%   B3:2/11  "HIGH OUTPUT PRESSURE OSR STORAGE BIT" %
%   B3:2/12  "HIGH OUTPUT PRESSURE OSR OUTPUT BIT" %
% Rung: 19 %
SOR BST XIC B3:2/12 NXB XIC B3:2/13 BND XIO B3:1/1 OTE B3:2/13 EOR
%   B3:2/12  "HIGH OUTPUT PRESSURE OSR OUTPUT BIT" %
%   B3:2/13  HI_OUT_FLOW_ALARM  "HIGH OUTPUT VALVE PRESSURE ALARM BIT" %
%   B3:1/1  ALARM_RESET  "ALRAM RESET PUSH BUTTON - HMI" %
% Rung: 20 %
SOR LES N7:3 10 XIC B3:0/5 XIC B3:0/15 XIO B3:1/1 BST TON T4:9 1.0 5 0 NXB XIC T4:9/DN OSR B3:2/14 B3:2/15 BND EOR
%   N7:3  OUTPUT_PRESSURE  "OUTPUT VALVE PRESSURE SCALED (0-100) PSI" %
%   B3:0/5  "OUTPUT PRESSURE BIT" %
%   B3:0/15  OUTPUT_VALVE_RELEASE  "OUTPUT VALVE RELEASE BIT" %
%   B3:1/1  ALARM_RESET  "ALRAM RESET PUSH BUTTON - HMI" %
%   T4:9  "LOW OUTPUT PRESSURE ALARM TIMER" %
%   T4:9/DN  "LOW OUTPUT PRESSURE TIMER DONE BIT" %
%   B3:2/14  "LOW OUTPT PRESSURE OSR STORAGE BIT" %
%   B3:2/15  "LOW OUTPUT PRESSURE OSR DONE BIT" %

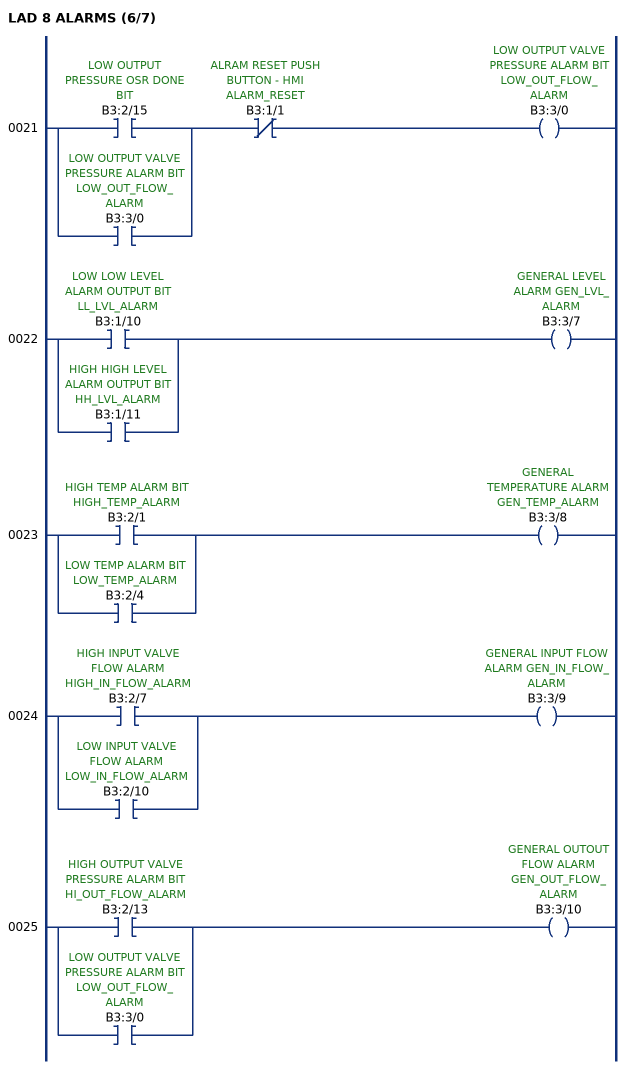
% Rung: 21 %
SOR BST XIC B3:2/15 NXB XIC B3:3/0 BND XIO B3:1/1 OTE B3:3/0 EOR
%   B3:2/15  "LOW OUTPUT PRESSURE OSR DONE BIT" %
%   B3:3/0  LOW_OUT_FLOW_ALARM  "LOW OUTPUT VALVE PRESSURE ALARM BIT" %
%   B3:1/1  ALARM_RESET  "ALRAM RESET PUSH BUTTON - HMI" %
% Rung: 22 %
SOR BST XIC B3:1/10 NXB XIC B3:1/11 BND OTE B3:3/7 EOR
%   B3:1/10  LL_LVL_ALARM  "LOW LOW LEVEL ALARM OUTPUT BIT" %
%   B3:1/11  HH_LVL_ALARM  "HIGH HIGH LEVEL ALARM OUTPUT BIT" %
%   B3:3/7  GEN_LVL_ALARM  "GENERAL LEVEL ALARM" %
% Rung: 23 %
SOR BST XIC B3:2/1 NXB XIC B3:2/4 BND OTE B3:3/8 EOR
%   B3:2/1  HIGH_TEMP_ALARM  "HIGH TEMP ALARM BIT" %
%   B3:2/4  LOW_TEMP_ALARM  "LOW TEMP ALARM BIT" %
%   B3:3/8  GEN_TEMP_ALARM  "GENERAL TEMPERATURE ALARM" %
% Rung: 24 %
SOR BST XIC B3:2/7 NXB XIC B3:2/10 BND OTE B3:3/9 EOR
%   B3:2/7  HIGH_IN_FLOW_ALARM  "HIGH INPUT VALVE FLOW ALARM" %
%   B3:2/10  LOW_IN_FLOW_ALARM  "LOW INPUT VALVE FLOW ALARM" %
%   B3:3/9  GEN_IN_FLOW_ALARM  "GENERAL INPUT FLOW ALARM" %
% Rung: 25 %
SOR BST XIC B3:2/13 NXB XIC B3:3/0 BND OTE B3:3/10 EOR
%   B3:2/13  HI_OUT_FLOW_ALARM  "HIGH OUTPUT VALVE PRESSURE ALARM BIT" %
%   B3:3/0  LOW_OUT_FLOW_ALARM  "LOW OUTPUT VALVE PRESSURE ALARM BIT" %
%   B3:3/10  GEN_OUT_FLOW_ALARM  "GENERAL OUTOUT FLOW ALARM" %

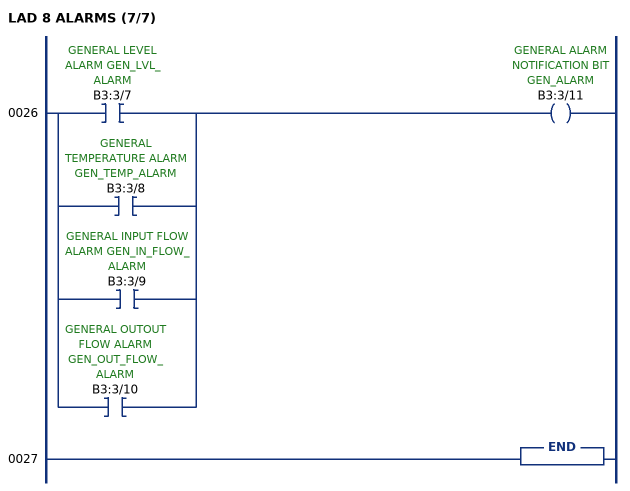
% Rung: 26 %
SOR BST XIC B3:3/7 NXB XIC B3:3/8 NXB XIC B3:3/9 NXB XIC B3:3/10 BND OTE B3:3/11 EOR
%   B3:3/7  GEN_LVL_ALARM  "GENERAL LEVEL ALARM" %
%   B3:3/8  GEN_TEMP_ALARM  "GENERAL TEMPERATURE ALARM" %
%   B3:3/9  GEN_IN_FLOW_ALARM  "GENERAL INPUT FLOW ALARM" %
%   B3:3/10  GEN_OUT_FLOW_ALARM  "GENERAL OUTOUT FLOW ALARM" %
%   B3:3/11  GEN_ALARM  "GENERAL ALARM NOTIFICATION BIT" %
% Rung: 27 %
SOR END EOR

LADDER 9 "DISPLAY"
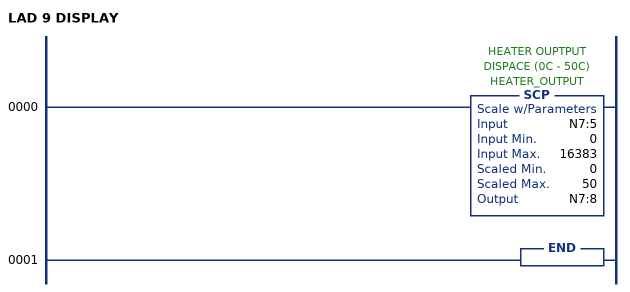
% Rung: 0 %
SOR SCP N7:5 0 16383 0 50 N7:8 EOR
%   N7:5  "HEATER CONTROL VARIABLE" %
%   N7:8  HEATER_OUTPUT  "HEATER OUPTPUT DISPACE (0C - 50C)" %
% Rung: 1 %
SOR END EOR

OTHER DOCUMENTED ADDRESSES
  B3:2/8  "LOW INPUT PRESSURE OSR STORAGE BIT"
  B3:3/13  "TANK DRAIN ONE SHOT"
  B3:3/14  "TANK DRAIN ONE SHOT"
  B3:4/5  "MAUNAL TANK DRAIN ONS"
  B3:4/6  "MANUAL TANK DRAIN TRIGGER"
  B3:4/9  "SYSTEM ERROR ONE SHOT"
  F8:0/0  "TANK LEVEL SENSOR FLOAT SCALED (0 - 100)%"
  N7:0/0  "SYSTEM STATUS 0 = OFF 1 = ON 2 = ERROR"
  N7:0/1  "HEATER STATUS 0 = OFF 1 = HAND 2 = AUTO"
  N7:0/2  "INPUT VALVE PRESSURE SCALED (0 - 100 PSI)"
  N7:0/3  "OUTPUT VALVE PRESSURE SCALED (0-100) PSI"
  N7:0/4  "THERMOCOUPLE INPUT INT SCALED (0C TO 50C)"
  N7:0/5  "HEATER CONTROL VARIABLE"
  N7:0/6  HMI_AUTO_TEMP_IN  "AUTO TEMPERATURE HMI INPUT"
  PD9:0.2  "AUTO TEMPERATURE CONTROL SCALED(0 - 16383) SET POINT"
  PFILE:3  "Digital Input ladder"
  T4:7/DN  "LOW INPUT PRESSURE TIMER DONE BIT"

REVISION NOTES
  1: All Done !

DATA TABLE (non-zero values as saved)
DATA T4
% .PRE .ACC %
% T4:0 % 10 0
% T4:1 % 10 0
% T4:2 % 10 0
% T4:3 % 10 0
% T4:4 % 300 0
% T4:5 % 300 0
% T4:6 % 5 0
% T4:7 % 5 0
% T4:8 % 5 0
% T4:9 % 5 0
% T4:10 % 15 0
% T4:11 % 15 0
% T4:12 % 10 0
